{attribute 'qualified_only'}
{attribute 'strict'}
TYPE E_HeightTest_State :
(
	//GENERIC

	READY				,
	//MANUAL_MODE			:=50, /manual mode not needed.
	ERROR				,
	//SPECIFIC FOR EVERY STATION
	MEASURE				,
	WAIT_MEASUREMENT	,
	DONE				,
	RESULTS				,
	RESET				
);
END_TYPE

(* stored: Version 1.1.0.1, ProductVersion 3.1.4024.13
   DUT E_HeightTest_State: Id {5ddfb4d9-7fc1-463c-94a3-7a2a15a0ec39} *)
